{attribute 'linkalways'} 
{attribute 'no_explicit_call' := 'This FB is a CLASS and must be accessed using methods or properties'}
{attribute 'enable_dynamic_creation'}
FUNCTION_BLOCK _ETcVnContourRetrievalMode EXTENDS EnumDatatypeBase
VAR
	localData : ETcVnContourRetrievalMode;
	activeData : REFERENCE TO ETcVnContourRetrievalMode;
	enumBaseDatatype : _DINT(localData);
END_VAR

METHOD PRIVATE AddLocalEnumeration
VAR_INPUT
	Enumeration : T_MAXSTRING;
	Value : ETcVnContourRetrievalMode;
END_VAR
AddEnumeration(Enumeration, Value);
END_METHOD

PROPERTY PUBLIC Address : PVOID
GET
Address := ADR(activeData);
END_GET
END_PROPERTY

METHOD PUBLIC ClearReference
VAR_INPUT
END_VAR
activeData REF= localData;
SetBaseDatatypeReference();
END_METHOD

METHOD PUBLIC Clone : I_Datatype
VAR
    pClone : POINTER TO _ETcVnContourRetrievalMode;
END_VAR
pClone := __NEW(_ETcVnContourRetrievalMode(InitialValue := Value));
Clone := pClone^;
END_METHOD

METHOD FB_init : BOOL
VAR_INPUT
	bInitRetains : BOOL; // if TRUE, the retain variables are initialized (warm start / cold start)
	bInCopyCode : BOOL;  // if TRUE, the instance afterwards gets moved into the copy code (online change)
	InitialValue : ETcVnContourRetrievalMode;
END_VAR
localData := InitialValue;
AddBaseDatatype(enumBaseDatatype);
ClearReference();

AddLocalEnumeration('TCVN_CRM_EXTERNAL', ETcVnContourRetrievalMode.TCVN_CRM_EXTERNAL);
AddLocalEnumeration('TCVN_CRM_LIST', ETcVnContourRetrievalMode.TCVN_CRM_LIST);
AddLocalEnumeration('TCVN_CRM_CONNECTED_COMPONENTS', ETcVnContourRetrievalMode.TCVN_CRM_CONNECTED_COMPONENTS);
AddLocalEnumeration('TCVN_CRM_TREE', ETcVnContourRetrievalMode.TCVN_CRM_TREE);
AddLocalEnumeration('TCVN_CRM_FLOODFILL', ETcVnContourRetrievalMode.TCVN_CRM_FLOODFILL);
END_METHOD

PROPERTY PUBLIC Identifier : T_MAXSTRING
GET
Identifier := 'ETcVnContourRetrievalMode';
END_GET
END_PROPERTY

METHOD IsEnumeratorValueEqual : BOOL
VAR_INPUT
	Enumerator : I_KeyValueForwardEnumerator;
END_VAR
VAR
	storedValue : ETcVnContourRetrievalMode;
END_VAR
IF NOT Enumerator.TryGet(storedValue) THEN
	RETURN;
END_IF

IsEnumeratorValueEqual := storedValue = activeData;
END_METHOD

METHOD PUBLIC MakeReferenceTo
VAR_INPUT
	ReferenceTarget : REFERENCE TO ETcVnContourRetrievalMode;
END_VAR
activeData REF= ReferenceTarget;
SetBaseDatatypeReference();
END_METHOD

METHOD PROTECTED SetBaseDatatypeReference
VAR_INPUT
END_VAR
enumBaseDatatype.MakeReferenceTo(activeData);
END_METHOD

PROPERTY PUBLIC Size : UDINT
GET
Size := SIZEOF(activeData);
END_GET
END_PROPERTY

METHOD TryMakeReferenceTo : BOOL
VAR_INPUT
	Target : I_Datatype;
END_VAR
VAR
	targetAsEnum : I_EnumDatatype;
	pTargetData : POINTER TO ETcVnContourRetrievalMode;
END_VAR
IF NOT Target.TryResolveAsEnumDatatype(targetAsEnum) THEN
	RETURN;
END_IF

IF targetAsEnum.Identifier <> Identifier THEN
	RETURN;
END_IF

pTargetData := Target.Address;
activeData REF= pTargetData^;
SetBaseDatatypeReference();
TryMakeReferenceTo := TRUE;
END_METHOD

PROPERTY PUBLIC Value : ETcVnContourRetrievalMode
GET
Value := activeData;
END_GET
SET
activeData := Value;
END_SET
END_PROPERTY

END_FUNCTION_BLOCK

(* stored: Version 1.1.0.1
   POU _ETcVnContourRetrievalMode: Id {1ea80a99-8cbb-413a-bde3-5b12c945882d}, SpecialFunc None
   Folder Constructor: Id {5de5becf-c784-4c2d-8dbe-6ee6ba419a55}
   Folder Private: Id {6358ea48-fd3c-42f1-87ac-019df987d474}
   Folder Protected: Id {2c7f1865-bb61-491d-9c51-0caee45692c9}
   Method AddLocalEnumeration: Id {9878676b-65ee-4ca9-8965-b967a4d36f9c}
   Property Address: Id {107a1bb2-0fec-4f7a-a9ac-b81750e174b5}
   Get Get: Id {ffadb304-e114-463e-b6ee-e296c12a30ec}
   Method ClearReference: Id {70d1e9a3-1c1f-45df-bce5-7f92f472e403}
   Method Clone: Id {49fbc892-760e-4326-b4f4-421c2c9ce386}
   Method FB_init: Id {eba1d857-7c63-4316-a113-3defac0887c3}
   Property Identifier: Id {7dd9a36c-fa85-4c8d-b920-27d31e8c8062}
   Get Get: Id {c1b3ed8d-afa8-4205-8d4b-de5a0b552b30}
   Method IsEnumeratorValueEqual: Id {502be19b-3d82-4993-b309-22880873f1a2}
   Method MakeReferenceTo: Id {5dc29a90-abbe-4d99-a9e9-49dbb85d9222}
   Method SetBaseDatatypeReference: Id {ce55a017-2372-4e54-905b-03c81b9b58ed}
   Property Size: Id {ab3278b6-a0d2-49d2-a065-5ea1ee1daa2c}
   Get Get: Id {f17539f3-bb04-40c9-8cd5-23cb3a75d82a}
   Method TryMakeReferenceTo: Id {2dcd8d85-8864-4200-aac0-08799efded3b}
   Property Value: Id {aeaa9d2f-cb10-43f1-9343-c1380f9522de}
   Get Get: Id {245bfe01-f18d-4818-bd8b-4682b5bd8a7b}
   Set Set: Id {b9ab1e7e-df60-4213-9b2c-cd97f7da859d} *)
